Fanuc KAREL source: NC0071.KL

-- PROVISIONAL review KL for V1013-1; original PC SHA256 e40067551157435479351246903c68435ebe7946ac714393e74ae6a2f2472219
-- Incomplete behavior may be omitted. Consult companion uncertainty JSON. Do not deploy.
PROGRAM NC0071
%NOLOCKGROUP
-- UNRESOLVED_LOCAL_POOL 21 cells at code offset 3; source declarations unknown
-- DIRECT_LOCAL_WORD_ACCESS alone does not prove INTEGER, REAL, or BOOLEAN
BEGIN
  -- UNRESOLVED_PC offsets 0-8; opcodes 2B,2C,7B
  -- UNRESOLVED_PC offsets 13-20; opcodes 9D,23
  -- UNRESOLVED_PC offsets 25-54; opcodes 9D,23,9E,2E,22,7A
  -- UNRESOLVED_PC offsets 59-88; opcodes 9D,23,9E,2E,22,7A
  -- UNRESOLVED_PC offsets 93-122; opcodes 9D,23,9E,2E,22,7A
  -- UNRESOLVED_PC offsets 127-156; opcodes 9D,23,9E,2E,22,7A
  -- UNRESOLVED_PC offsets 161-190; opcodes 9D,23,9E,2E,22,7A
  -- UNRESOLVED_PC offsets 195-224; opcodes 9D,23,9E,2E,22,7A
  -- UNRESOLVED_PC offsets 229-258; opcodes 9D,23,9E,2E,22,7A
  -- UNRESOLVED_PC offsets 263-292; opcodes 9D,23,9E,2E,22,7A
  -- UNRESOLVED_PC offsets 297-326; opcodes 9D,23,9E,2E,22,7A
  -- UNRESOLVED_PC offsets 331-360; opcodes 9D,23,9E,2E,22,7A
  -- UNRESOLVED_PC offsets 365-394; opcodes 9D,23,9E,2E,22,7A
  -- UNRESOLVED_PC offsets 399-428; opcodes 9D,23,9E,2E,22,7A
  -- UNRESOLVED_PC offsets 433-462; opcodes 9D,23,9E,2E,22,7A
  -- UNRESOLVED_PC offsets 467-496; opcodes 9D,23,9E,2E,22,7A
  -- UNRESOLVED_PC offsets 501-530; opcodes 9D,23,9E,2E,22,7A
  -- UNRESOLVED_PC offsets 535-564; opcodes 9D,23,9E,2E,22,7A
  -- UNRESOLVED_PC offsets 569-598; opcodes 9D,23,9E,2E,22,7A
  -- UNRESOLVED_PC offsets 603-632; opcodes 9D,23,9E,2E,22,7A
  -- UNRESOLVED_PC offsets 637-666; opcodes 9D,23,9E,2E,22,7A
  -- UNRESOLVED_PC offsets 671-700; opcodes 9D,23,9E,2E,22,7A
  -- UNRESOLVED_PC offsets 705-719; opcodes 21,9D,52,23
  -- UNRESOLVED_PC offsets 724-739; opcodes 20,2C,23
  -- UNRESOLVED_PC offsets 744-759; opcodes 20,2C,23
  -- UNRESOLVED_PC offsets 764-779; opcodes 20,2C,23
  -- UNRESOLVED_PC offsets 784-799; opcodes 20,2C,23
  -- UNRESOLVED_PC offsets 804-819; opcodes 20,2C,23
  -- UNRESOLVED_PC offsets 824-839; opcodes 20,2C,23
  -- UNRESOLVED_PC offsets 844-859; opcodes 20,2C,23
  -- UNRESOLVED_PC offsets 864-879; opcodes 20,2C,23
  -- UNRESOLVED_PC offsets 884-899; opcodes 20,2C,23
  -- UNRESOLVED_PC offsets 904-919; opcodes 20,2C,23
  -- UNRESOLVED_PC offsets 924-939; opcodes 20,2C,23
  -- UNRESOLVED_PC offsets 944-959; opcodes 20,2C,23
  -- UNRESOLVED_PC offsets 964-979; opcodes 20,2C,23
  -- UNRESOLVED_PC offsets 984-999; opcodes 20,2C,23
  -- UNRESOLVED_PC offsets 1004-1019; opcodes 20,2C,23
  -- UNRESOLVED_PC offsets 1024-1039; opcodes 20,2C,23
  -- UNRESOLVED_PC offsets 1044-1059; opcodes 20,2C,23
  -- UNRESOLVED_PC offsets 1064-1079; opcodes 20,2C,23
  -- UNRESOLVED_PC offsets 1084-1099; opcodes 20,2C,23
  -- UNRESOLVED_PC offsets 1104-1119; opcodes 20,2C,23
  -- UNRESOLVED_PC offsets 1124-1128; opcodes 7F
  -- UNRESOLVED_PC offsets 1133-1137; opcodes 27,AA
  -- UNRESOLVED_PC offsets 1142-1146; opcodes 7F
END NC0071
